# EPICS autosave request: optics/opticsApp/Db/filterDrive.req
$(P)$(R)TransmissionSetpoint
$(P)$(R)FilterMaskSetpoint
$(P)$(R)EnergySelect
$(P)$(R)EnergyLocal
$(P)$(R)WaitTime
$(P)$(R)Debug
